TYPE ACRMemoryUDIntEvent EXTENDS ACRMemoryEvent :
STRUCT
	_Value : UDINT;
END_STRUCT
END_TYPE

(* stored: Version 1.1.0.1, ProductVersion 3.1.4020.12
   DUT ACRMemoryUDIntEvent: Id {9cf96008-7017-41b0-bcb1-4ae7bde398bb} *)
